// TIA Portal V19 export
DATA_BLOCK "SUGAR DB"   // DB162
{ S7_Optimized_Access := 'TRUE' }
// stored: MemoryReserve 100
   VAR
      START : Bool;
   END_VAR
   VAR RETAIN
      PAUSE : Bool;
   END_VAR
   VAR
      STOP : Bool;
   END_VAR
   VAR RETAIN
      "AUTO BUFF" : Int;
   END_VAR
   VAR
      "SUGAR PROCESS OVER" : Bool;
      BIT : Struct
         "PURIFIED WATER" : Struct
            "PURIFIED WATER SELECT" : Bool;
            "PURIFIED WATER SKIP" : Bool;
            "PURIFIED WATER PROCESS OF INITIAL DRAIN SELECT" : Bool;
            "PURIFIED WATER PROCESS OF INITIAL DRAIN SKIP" : Bool;
            "PURIFIED WATER LOAD CELL" : Bool;
            "SELECT HEATING" : Bool;
            "PURIFIED WATER OVER" : Bool;
            "PURIFIED WATER PROCESS OF JACKET DRAIN SELECT" : Bool;
            "PURIFIED WATER PROCESS OF JACKET DRAIN SKIP" : Bool;
         END_STRUCT;
         "MATERIAL SUCTION" : Struct
            "MATERIAL SUCTION SELECT" : Bool;
            "MATERIAL SUCTION SKIP" : Bool;
            "MATERIAL SUCTION OVER" : Bool;
         END_STRUCT;
      END_STRUCT;
   END_VAR
   VAR RETAIN
      "SET PARAMETER" : Struct
         "PURIFIED WATER INITIAL DRAIN TIME" : Int;
         "PURIFIED LOAD" : Real;
         "PURIFIED HEATING" : Real;
         "PURIFIED COOLING" : Real;
         "PURIFIED STIRRER MOTOR RPM" : Real;
         "PURIFIED STIRRER_TIME" : Int;
         "PURIFIED WATER JACKET DRAIN TIME" : Int;
         "MATERIAL_SORBITOL LOAD CELL" : Real;
         "MATERIAL_SORBITOL STIRRER TIME" : Int;
         "MATERIAL SORBITOL STIRRER MOTOR RPM" : Real;
         "MATERIAL_SORBITOL TEMP_MAX" : Real;
         "MATERIAL_SORBITOL TEMP_MIN" : Real;
         "MATERIAL_GLUCOSE LOAD CELL" : Real;
         "MATERIAL_GLUCOSE STIRRER TIME" : Int;
         "MATERIAL GLUCOSE STIRRER MOTOR RPM" : Real;
         "MATERIAL_GLUCOSE TEMP_MAX" : Real;
         "MATERIAL_GLUCOSE TEMP_MIN" : Real;
         "RECIRCULATION TOTAL TIME" : Int;
         "RECIRCULATION STIRRER RPM" : Real;
         "RECIRCULATION HOMOGENIZER DELAY" : Int;
         "MATERIAL SUCTION VACUUM HIGH" : Real;
         "MATERIAL SUCTION VACUUM LOW" : Real;
         "MATERIAL SUCTION STIRRER RPM" : Real;
         "MATERIAL SUCTION LOAD CELL" : Real;
      END_STRUCT;
      "PV PARAMETER" : Struct
         "PURIFIED WATER INITIAL DRAIN TIME" : Int;
         "PURIFIED STIRRER_TIME" : Int;
         "PURIFIED WATER JACKET DRAIN TIME" : Int;
         "MATERIAL_SORBITOL STIRRER TIME" : Int;
         "MATERIAL_GLUCOSE STIRRER TIME" : Int;
         "RECIRCULATION TOTAL TIME" : Int;
         "RECIRCULATION HOMOGENIZER DELAY" : Int;
         "PURIFIED LOAD" : Real;
         "MATERIAL_SORBITOL LOAD CELL" : Real;
         "MATERIAL_GLUCOSE LOAD CELL" : Real;
         "MATERIAL SUCTION LOAD CELL" : Real;
      END_STRUCT;
   END_VAR
BEGIN
END_DATA_BLOCK
